KUKA KRL data list: check_dock_an.dat

&ACCESS RVO1
&REL 71
&COMMENT MB-CHECK_CONDITIONS_AN
&PARAM DISKPATH = KRC:\R1\TP
DEFDAT Check_dock_AN PUBLIC
;date:2012-08-14
ENDDAT
